FUNCTION_BLOCK FB_mqtt_publish IMPLEMENTS  ITF_CoeSdoEventHandler
VAR_INPUT
END_VAR
VAR_OUTPUT
END_VAR
VAR
	// published message
	fbMqttClient : FB_IotMqttClient;
	fbMessageQueue : FB_IotMqttMessageQueue;
	bSetParameter : BOOL := TRUE;
	bConnect : BOOL := TRUE;
	hrErrorOccurred : HRESULT; // contains the latest occurred error
	
	fbSerializer :FB_Serializer;
	
	sTopicPub : STRING(255) := 'devices/unit230/messages/events/';
	
	// for making publish event
	publish_cycle_timer :TON;
	datetime_string: STRING(39);
	
	publish_command: BOOL;
	_error_id :UDINT;
	
END_VAR


// Connect MQTT broker and publish

IF bSetParameter THEN
	bSetParameter := FALSE;
	fbMqttClient.sHostName := 'IndustrialOPNFair2024-IoTHub.azure-devices.net';
	fbMqttClient.nHostPort := 8883;
	fbMqttClient.stTLS.sCA := 'c:\TwinCAT\3.1\Config\Certificates\BaltimoreCyberTrust.cer'; // CA certificate 
	fbMqttClient.sClientId := 'unit230';
	fbMqttClient.stTLS.sAzureSas := 'HostName=IndustrialOPNFair2024-IoTHub.azure-devices.net;DeviceId=unit230;SharedAccessSignature=SharedAccessSignature sr=IndustrialOPNFair2024-IoTHub.azure-devices.net%2Fdevices%2Funit230&sig=aZHGqBLbPbZ0nCj3%2BrwgAJAAhzI2BvVoTXPMA%2BaobPA%3D&se=1734308970'; // Device SAS Token
	fbMqttClient.stTLS.bNoServerCertCheck:=TRUE;
	(*
	//fbMqttClient.stTLS.sCA := 'c:\TwinCAT\3.1\Config\Certificates\BaltimoreCyberTrust.crt'; // CA certificate 
	//fbMqttClient.stTLS.sAzureSas := 'HostName=IndustrialOPNFair2024-IoTHub.azure-devices.net;DeviceId=unit230;SharedAccessSignature=SharedAccessSignature sr=IndustrialOPNFair2024-IoTHub.azure-devices.net%2Fdevices%2Funit230&sig=GxT9x70t1Q1per9XXu4Az%2FJhK1jBZt14KJ%2B7LG4NB%2Fw%3D&se=1712921181'; // Device SAS Token
	fbMqttClient.sClientId := 'unit230';
	fbMqttClient.sHostName := '192.168.1.20';
	fbMqttClient.nHostPort := 1883;
	*)
	fbMqttClient.ipMessageQueue := fbMessageQueue;
END_IF

fbMqttClient.Execute(bConnect);
IF fbMqttClient.bError THEN
  // add your error logging here
  hrErrorOccurred := fbMqttClient.hrErrorCode;
END_IF


publish_cycle_timer(IN := NOT publish_command, PT := T#5S);

IF publish_cycle_timer.Q THEN
	publish_command := TRUE;
END_IF

{warning 'add property implementation'}
PROPERTY nErrID : UDINT
GET
nErrID := _error_id;
END_GET
END_PROPERTY

{warning 'add method implementation '}
METHOD sdo_data_received : BOOL
VAR_INPUT
	command	: REFERENCE TO bajp_diagtool.CoeSdoCommand;
END_VAR
VAR
	diag_data_body: POINTER TO sdo_xplanar_aps_diag;
	temp: UDINT;
	i: UINT;
END_VAR
VAR_INST
		tile_number : UINT;
		sPayloadPub : STRING(255);
		pub_complete : ARRAY [1..2] OF BOOL;
END_VAR
diag_data_body := command.pDstBuf;
CASE command.nSlaveAddr OF
	1001:
		tile_number := 1;
	1003:
		tile_number := 2;
END_CASE

IF publish_command AND fbMqttClient.bConnected THEN
	datetime_string := SYSTEMTIME_TO_ISO8601(
		systemTime := command.datetime,
		nBias := 0,
		bUTC := TRUE,
		nPrecision := 3
	);
	CASE tile_number OF
		1:
			temp := diag_data_body^.temperature_west;
		2:
			temp := diag_data_body^.temperature_east;
	END_CASE
	sPayloadPub := fbSerializer.serialize(
	  datetime := datetime_string,
	  device_name := CONCAT('xplanar_tile_', UINT_TO_STRING(tile_number)),
	  temp := temp,
	  fan_rpm := diag_data_body^.fan_rpm,
	  current := diag_data_body^.power_supply_current
	);
	IF fbMqttClient.Publish(	sTopic:= sTopicPub, 
				pPayload:= ADR(sPayloadPub), nPayloadSize:= LEN2(ADR(sPayloadPub)), 
				eQoS:= TcIotMqttQos.AtMostOnceDelivery, bRetain:= FALSE, bQueue:= FALSE ) THEN
		_error_id := 0;
		sdo_data_received := TRUE;
	END_IF
    IF fbMqttClient.bError THEN
      // add your error logging here
    	_error_id := TO_UDINT(fbMqttClient.hrErrorCode);
	  	sdo_data_received := TRUE;
	ELSE
		pub_complete[tile_number] := TRUE;
    END_IF
	publish_command := FALSE;
	FOR i := 1 TO 2 DO
		IF NOT pub_complete[i] THEN
			publish_command := TRUE;
		END_IF
	END_FOR
ELSE
	FOR i := 1 TO 2 DO
		pub_complete[i] := FALSE;
	END_FOR
END_IF
END_METHOD

END_FUNCTION_BLOCK

(* stored: Version 1.1.0.1, ProductVersion 3.1.4024.12
   POU FB_mqtt_publish: Id {1aff89c1-b24e-4329-a407-cdf41e6202bf}, SpecialFunc None
   Property nErrID: Id {23e231bd-c44f-4e02-8a8b-e9645fc01229}
   Get Get: Id {91a8df65-1b9a-4afb-bfdf-be827636d678}
   Method sdo_data_received: Id {598e3abe-0bfd-47c5-95e4-1fd355927e50} *)
